TYPE U32 : UDINT; END_TYPE

(* stored: Version 1.1.0.1
   DUT U32: Id {6b7c6099-38f9-0a0c-13f9-ad2c1a6a91bd} *)
